PROGRAM EventLogger
VAR CONSTANT
	uiNumberOfAlarms 		: WORD := 1000;
END_VAR
VAR
	a_fbEventAlarm			: ARRAY [0..uiNumberOfAlarms] OF fb_EventAlarm;
	w_index					: WORD;
	
END_VAR
VAR // added by the converter: edge detectors and wires of the graphical bodies
    _w1, _w2, _w3, _w8 : ANY;
    _w4, _w5, _w6, _w7 : BOOL;
END_VAR

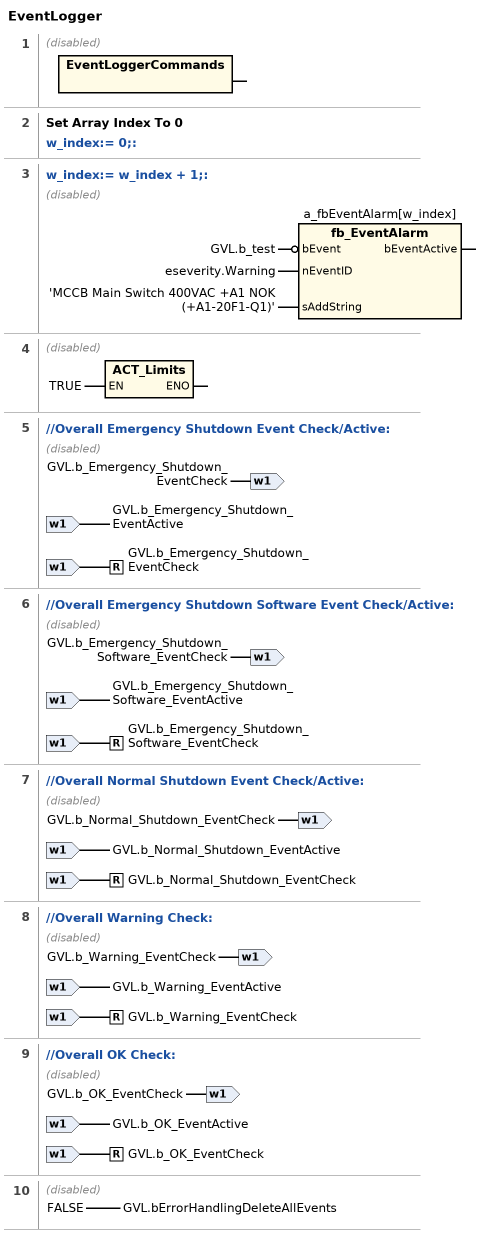
// NETWORK 1 (disabled)
// EventLoggerCommands();

// NETWORK 2: Set Array Index To 0
// label: w_index:= 0;

// NETWORK 3 (disabled)
// label: w_index:= w_index + 1;
// a_fbEventAlarm[w_index](
//     bEvent := NOT GVL.b_test,
//     nEventID := eseverity.Warning,
//     sAddString := 'MCCB Main Switch 400VAC +A1 NOK (+A1-20F1-Q1)'); // fb_EventAlarm

// NETWORK 4 (disabled)
// ACT_Limits();

// NETWORK 5 (disabled)
// label: //Overall Emergency Shutdown Event Check/Active
// _w1 := GVL.b_Emergency_Shutdown_EventCheck;
// GVL.b_Emergency_Shutdown_EventActive := _w1;
// GVL.b_Emergency_Shutdown_EventCheck R= _w1;

// NETWORK 6 (disabled)
// label: //Overall Emergency Shutdown Software Event Check/Active
// _w2 := GVL.b_Emergency_Shutdown_Software_EventCheck;
// GVL.b_Emergency_Shutdown_Software_EventActive := _w2;
// GVL.b_Emergency_Shutdown_Software_EventCheck R= _w2;

// NETWORK 7 (disabled)
// label: //Overall Normal Shutdown Event Check/Active
// _w3 := GVL.b_Normal_Shutdown_EventCheck;
// GVL.b_Normal_Shutdown_EventActive := _w3;
// GVL.b_Normal_Shutdown_EventCheck R= _w3;

// NETWORK 8 (disabled)
// label: //Overall Warning Check
// _w4 := GVL.b_Warning_EventCheck;
// GVL.b_Warning_EventActive := _w4;
// GVL.b_Warning_EventCheck R= _w4;

// NETWORK 9 (disabled)
// label: //Overall OK Check
// _w5 := GVL.b_OK_EventCheck;
// GVL.b_OK_EventActive := _w5;
// GVL.b_OK_EventCheck R= _w5;

// NETWORK 10 (disabled)
// GVL.bErrorHandlingDeleteAllEvents := FALSE;

ACTION ACT_Limits:
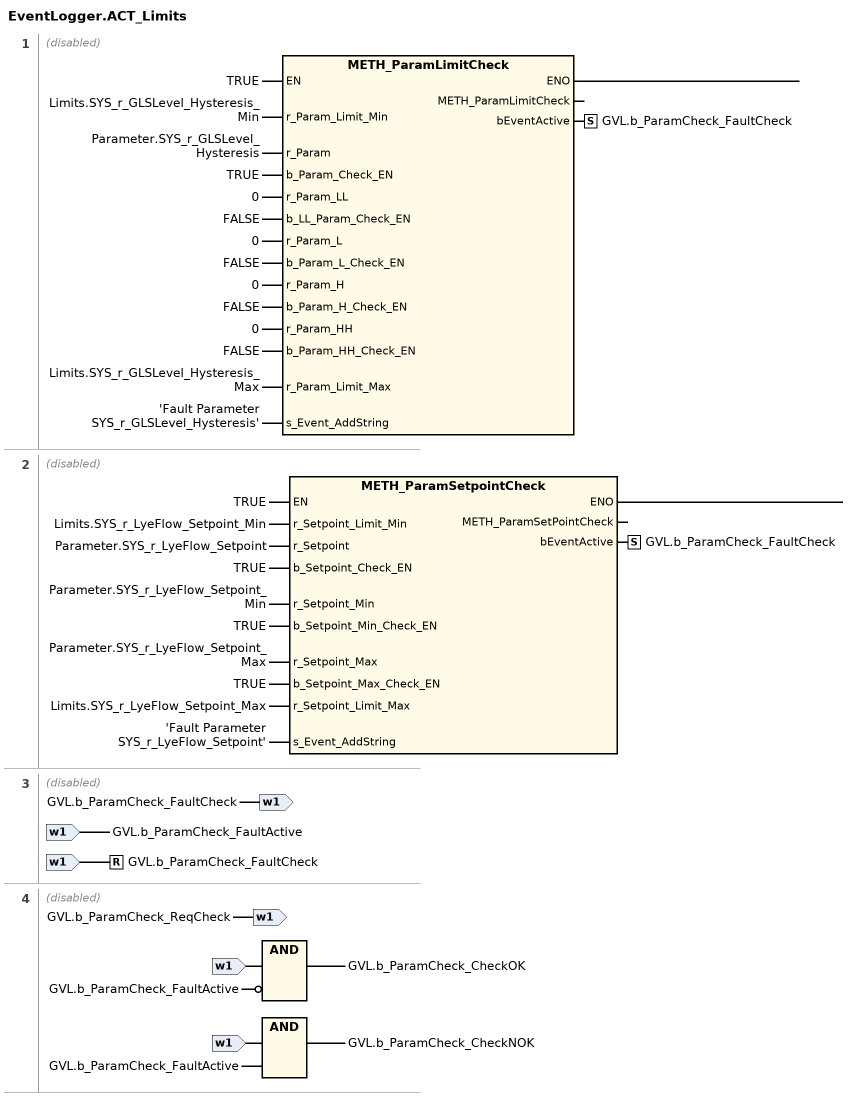
// NETWORK 1 (disabled)
// METH_ParamLimitCheck(r_Param_Limit_Min := Limits.SYS_r_GLSLevel_Hysteresis_Min, r_Param := Parameter.SYS_r_GLSLevel_Hysteresis, b_Param_Check_EN := TRUE, r_Param_LL := 0, b_LL_Param_Check_EN := FALSE, r_Param_L := 0, b_Param_L_Check_EN := FALSE, r_Param_H := 0, b_Param_H_Check_EN := FALSE, r_Param_HH := 0, b_Param_HH_Check_EN := FALSE, r_Param_Limit_Max := Limits.SYS_r_GLSLevel_Hysteresis_Max, s_Event_AddString := 'Fault Parameter SYS_r_GLSLevel_Hysteresis', bEventActive => _w6);
// GVL.b_ParamCheck_FaultCheck S= _w6;

// NETWORK 2 (disabled)
// METH_ParamSetpointCheck(r_Setpoint_Limit_Min := Limits.SYS_r_LyeFlow_Setpoint_Min, r_Setpoint := Parameter.SYS_r_LyeFlow_Setpoint, b_Setpoint_Check_EN := TRUE, r_Setpoint_Min := Parameter.SYS_r_LyeFlow_Setpoint_Min, b_Setpoint_Min_Check_EN := TRUE, r_Setpoint_Max := Parameter.SYS_r_LyeFlow_Setpoint_Max, b_Setpoint_Max_Check_EN := TRUE, r_Setpoint_Limit_Max := Limits.SYS_r_LyeFlow_Setpoint_Max, s_Event_AddString := 'Fault Parameter SYS_r_LyeFlow_Setpoint', bEventActive => _w7);
// GVL.b_ParamCheck_FaultCheck S= _w7;

// NETWORK 3 (disabled)
// _w8 := GVL.b_ParamCheck_FaultCheck;
// GVL.b_ParamCheck_FaultActive := _w8;
// GVL.b_ParamCheck_FaultCheck R= _w8;

// NETWORK 4 (disabled)
// GVL.b_ParamCheck_CheckOK := GVL.b_ParamCheck_ReqCheck AND NOT GVL.b_ParamCheck_FaultActive;
// GVL.b_ParamCheck_CheckNOK := GVL.b_ParamCheck_ReqCheck AND GVL.b_ParamCheck_FaultActive;
END_ACTION

METHOD METH_ParamLimitCheck : BOOL
VAR_INPUT
	r_Param_Limit_Min			: REAL;
	r_Param				: REAL;
	b_Param_Check_EN	: BOOL;
	r_Param_LL 			: REAL;
	b_LL_Param_Check_EN : BOOL;
	r_Param_L 			: REAL;
	b_Param_L_Check_EN 	: BOOL;
	r_Param_H 			: REAL;
	b_Param_H_Check_EN 	: BOOL;
	r_Param_HH 			: REAL;
	b_Param_HH_Check_EN 	: BOOL;
	r_Param_Limit_Max 			: REAL ;
	s_Event_AddString : STRING;
END_VAR
VAR_OUTPUT
	bEventActive 				: BOOL;
END_VAR
bEventActive:=FALSE;

IF b_Param_Check_EN THEN
	//Fault when Param < Minimum
	w_index:= w_index + 1;
	a_fbEventAlarm[w_index](
		bEvent:=r_Param < r_Param_Limit_Min,
		nEventID:=eseverity.NormalShutdown,
		sAddString:=CONCAT(s_Event_AddString,' < Min-Value!'),
		bEventActive=>
	);
	IF a_fbEventAlarm[w_index].bEventActive THEN bEventActive := TRUE; END_IF;
		
	//Fault when Param > Maximum
	w_index:= w_index + 1;
	a_fbEventAlarm[w_index](
		bEvent:=r_Param > r_Param_Limit_Max,
		nEventID:=eseverity.NormalShutdown,
		sAddString:=CONCAT(s_Event_AddString,' > Max-Value!'),
		bEventActive=>
	);
	IF a_fbEventAlarm[w_index].bEventActive THEN bEventActive := TRUE; END_IF
END_IF

IF b_LL_Param_Check_EN THEN
	//Fault when Param_LL < Minimum
	w_index:= w_index + 1;
	a_fbEventAlarm[w_index](
		bEvent:=r_Param_LL < r_Param_Limit_Min,
		nEventID:=eseverity.NormalShutdown,
		sAddString:=CONCAT(s_Event_AddString,'_LL < Min-Value!'),
		bEventActive=>
	);
	IF a_fbEventAlarm[w_index].bEventActive THEN bEventActive := TRUE; END_IF;
		
	//Fault when Param_LL > Maximum
	w_index:= w_index + 1;
	a_fbEventAlarm[w_index](
		bEvent:=r_Param_LL > r_Param_Limit_Max,
		nEventID:=eseverity.NormalShutdown,
		sAddString:=CONCAT(s_Event_AddString,'_LL > Max-Value!'),
		bEventActive=>
	);
	IF a_fbEventAlarm[w_index].bEventActive THEN bEventActive := TRUE; END_IF
END_IF

IF b_Param_L_Check_EN THEN
	//Fault when Param_L < Minimum
	w_index:= w_index + 1;
	a_fbEventAlarm[w_index](
		bEvent:=r_Param_L < r_Param_Limit_Min,
		nEventID:=eseverity.NormalShutdown,
		sAddString:=CONCAT(s_Event_AddString,'_L < Min-Value!'),
		bEventActive=>
	);
	IF a_fbEventAlarm[w_index].bEventActive THEN bEventActive := TRUE; END_IF
	
	//Fault when Param_L > Maximum
	w_index:= w_index + 1;
	a_fbEventAlarm[w_index](
		bEvent:=r_Param_L > r_Param_Limit_Max,
		nEventID:=eseverity.NormalShutdown,
		sAddString:=CONCAT(s_Event_AddString,'_L > Max-Value!'),
		bEventActive=>
	);
END_IF

IF b_Param_H_Check_EN THEN
	//Fault when Param_H < Minimum
	w_index:= w_index + 1;
	a_fbEventAlarm[w_index](
		bEvent:=r_Param_H < r_Param_Limit_Min,
		nEventID:=eseverity.NormalShutdown,
		sAddString:=CONCAT(s_Event_AddString,'_H < Min-Value!'),
		bEventActive=>
	);
	IF a_fbEventAlarm[w_index].bEventActive THEN bEventActive := TRUE; END_IF
	
	//Fault when Param_H > Maximum
	w_index:= w_index + 1;
	a_fbEventAlarm[w_index](
		bEvent:=r_Param_H > r_Param_Limit_Max,
		nEventID:=eseverity.NormalShutdown,
		sAddString:=CONCAT(s_Event_AddString,'_H > Max-Value!'),
		bEventActive=>
	);
	IF a_fbEventAlarm[w_index].bEventActive THEN bEventActive := TRUE; END_IF
END_IF

IF b_Param_HH_Check_EN THEN
	//Fault when Param_HH < Minimum
	w_index:= w_index + 1;
	a_fbEventAlarm[w_index](
		bEvent:=r_Param_HH < r_Param_Limit_Min,
		nEventID:=eseverity.NormalShutdown,
		sAddString:=CONCAT(s_Event_AddString,'_HH < Min-Value!'),
		bEventActive=>
	);
	IF a_fbEventAlarm[w_index].bEventActive THEN bEventActive := TRUE; END_IF
	
	//Fault when Param_HH > Maximum
	w_index:= w_index + 1;
	a_fbEventAlarm[w_index](
		bEvent:=r_Param_HH > r_Param_Limit_Max,
		nEventID:=eseverity.NormalShutdown,
		sAddString:=CONCAT(s_Event_AddString,'_HH > Max-Value!'),
		bEventActive=>
	);
	IF a_fbEventAlarm[w_index].bEventActive THEN bEventActive := TRUE; END_IF
END_IF
END_METHOD

METHOD METH_ParamSetPointCheck 	: BOOL
VAR_INPUT
	r_Setpoint_Limit_Min		: REAL;
	r_Setpoint					: REAL;
	b_Setpoint_Check_EN			: BOOL;
	r_Setpoint_Min 				: REAL;
	b_Setpoint_Min_Check_EN 	: BOOL;
	r_Setpoint_Max 				: REAL;
	b_Setpoint_Max_Check_EN 	: BOOL;
	r_Setpoint_Limit_Max 		: REAL ;
	s_Event_AddString 			: STRING;
END_VAR
VAR_OUTPUT
	bEventActive 				: BOOL;
END_VAR
bEventActive:=FALSE;

IF b_Setpoint_Check_EN THEN
	//Fault when Param < Minimum
	w_index:= w_index + 1;
	a_fbEventAlarm[w_index](
		bEvent:=r_Setpoint < r_Setpoint_Limit_Min,
		nEventID:=eseverity.NormalShutdown,
		sAddString:=CONCAT(s_Event_AddString,' < Min-Value!'),
		bEventActive=>
	);
	IF a_fbEventAlarm[w_index].bEventActive THEN bEventActive := TRUE; END_IF;
		
	//Fault when Param > Maximum
	w_index:= w_index + 1;
	a_fbEventAlarm[w_index](
		bEvent:=r_Setpoint > r_Setpoint_Limit_Max,
		nEventID:=eseverity.NormalShutdown,
		sAddString:=CONCAT(s_Event_AddString,' > Max-Value!'),
		bEventActive=>
	);
	IF a_fbEventAlarm[w_index].bEventActive THEN bEventActive := TRUE; END_IF
END_IF

IF b_Setpoint_Min_Check_EN THEN
	//Fault when Param_LL < Minimum
	w_index:= w_index + 1;
	a_fbEventAlarm[w_index](
		bEvent:=r_Setpoint_Min < r_Setpoint_Limit_Min,
		nEventID:=eseverity.NormalShutdown,
		sAddString:=CONCAT(s_Event_AddString,'_Min < Min-Value!'),
		bEventActive=>
	);
	IF a_fbEventAlarm[w_index].bEventActive THEN bEventActive := TRUE; END_IF;
		
	//Fault when Param_Min > Maximum
	w_index:= w_index + 1;
	a_fbEventAlarm[w_index](
		bEvent:=r_Setpoint_Min > r_Setpoint_Limit_Max,
		nEventID:=eseverity.NormalShutdown,
		sAddString:=CONCAT(s_Event_AddString,'_Min > Max-Value!'),
		bEventActive=>
	);
	IF a_fbEventAlarm[w_index].bEventActive THEN bEventActive := TRUE; END_IF
END_IF

IF b_Setpoint_Max_Check_EN THEN
	//Fault when Param_Max < Minimum
	w_index:= w_index + 1;
	a_fbEventAlarm[w_index](
		bEvent:=r_Setpoint_Max < r_Setpoint_Limit_Min,
		nEventID:=eseverity.NormalShutdown,
		sAddString:=CONCAT(s_Event_AddString,'_Max < Min-Value!'),
		bEventActive=>
	);
	IF a_fbEventAlarm[w_index].bEventActive THEN bEventActive := TRUE; END_IF
	
	//Fault when Param_Max > Maximum
	w_index:= w_index + 1;
	a_fbEventAlarm[w_index](
		bEvent:=r_Setpoint_Max > r_Setpoint_Limit_Max,
		nEventID:=eseverity.NormalShutdown,
		sAddString:=CONCAT(s_Event_AddString,'_Max > Max-Value!'),
		bEventActive=>
	);
	IF a_fbEventAlarm[w_index].bEventActive THEN bEventActive := TRUE; END_IF
END_IF
END_METHOD

METHOD METH_ParamTimeCheck 	: BOOL
VAR_INPUT
	r_Time_Limit_Min		: TIME;
	r_Time					: TIME;
	r_Time_Limit_Max 		: TIME ;
	s_Event_AddString 		: STRING;
END_VAR
VAR_OUTPUT
	bEventActive 			: BOOL;
END_VAR
bEventActive:=FALSE;

//Fault when Time < Minimum
w_index:= w_index + 1;
a_fbEventAlarm[w_index](
	bEvent:=r_Time < r_Time_Limit_Min,
	nEventID:=eseverity.NormalShutdown,
	sAddString:=CONCAT(s_Event_AddString,' < Min-Value!'),
	bEventActive=>
);
IF a_fbEventAlarm[w_index].bEventActive THEN bEventActive := TRUE; END_IF;
	
//Fault when Time > Maximum
w_index:= w_index + 1;
a_fbEventAlarm[w_index](
	bEvent:=r_Time > r_Time_Limit_Max,
	nEventID:=eseverity.NormalShutdown,
	sAddString:=CONCAT(s_Event_AddString,' > Max-Value!'),
	bEventActive=>
);
IF a_fbEventAlarm[w_index].bEventActive THEN bEventActive := TRUE; END_IF
END_METHOD

END_PROGRAM

(* stored: Version 1.1.0.1, ProductVersion 3.1.4024.12
   POU EventLogger: Id {2a3b5e3f-2f78-4298-aad2-a68225e74544}, SpecialFunc None
   Action ACT_Limits: Id {3df82db2-97b6-455a-a3cd-3166a4dc9407}
   Method METH_ParamLimitCheck: Id {4c33c397-d204-456d-959b-1cc92452ef3f}
   Method METH_ParamSetPointCheck: Id {c6bf7ec2-ca7f-4f8c-9e73-b2db7de8e20c}
   Method METH_ParamTimeCheck: Id {171d5c75-147e-42dd-b239-fead585fea31} *)
